FUNCTION_BLOCK SEPARATION
VAR_INPUT
END_VAR
VAR_OUTPUT
END_VAR
VAR
END_VAR

END_FUNCTION_BLOCK

(* stored: Version 1.1.0.1, ProductVersion 3.1.4024.12
   POU SEPARATION: Id {742462ac-1e27-4045-b59f-5171acd4e492}, SpecialFunc None *)
